// TIA Portal V15.1 export
// export: Created 2024-06-21T08:40:57.1284392Z, ExportSetting WithDefaults, DisplayName Totally Integrated Automation Portal, DisplayVersion V15.1 Update 5, DisplayName TIA Portal Openness, DisplayVersion V15.1 Update 5, DisplayName SINAMICS Startdrive Advanced, DisplayVersion V15.1, DisplayName G130, G150, S120, S150, SINAMICS MV, S210, DisplayVersion V15.1, DisplayName G110M, G120, G120C, G120D, G120P, DisplayVersion V15.1, DisplayName STEP 7 Professional, DisplayVersion V15.1 Update 5, DisplayName STEP 7 Safety, DisplayVersion V15.1, DisplayName WinCC Professional, DisplayVersion V15.1 Update 5, DisplayName SIMATIC Visualization Architect, DisplayVersion V15.1
FUNCTION_BLOCK "L1SafetyFbkAlarm"   // FB1422, FBD
TITLE = L1SafetyFbkAlarm
{ S7_Optimized_Access := 'FALSE' }
AUTHOR : VCC
FAMILY : AlarmHnd
NAME : 1SafeAlm
VERSION : 0.3
// ================================================================================
// TThis module evalute the diagnostic byte from the Siemens safety Functionblock 
// FB 216 "F_FDBACK" and generates a feedback alarm in the standard program.
// A boolean output is available to inform the upper level that the alarm can be 
// reset.
// This module generates also a word containing all necessary information for HMI 
// Icon animation, and a word with all information for HMI safety module 
// diagnostic screen. 
// ================================================================================
// stored: AutoNumber false, IsIECCheckEnabled false, SetENOAutomatically False, UDAEnableTagReadback false
   VAR_INPUT
      I_Feedback { ExternalAccessible := 'False'; ExternalVisible := 'False'; ExternalWritable := 'False'} : Bool;   // Input feedback
      I_AlarmClass { ExternalAccessible := 'False'; ExternalVisible := 'False'; ExternalWritable := 'False'} : Char;   // Alarm class -> A - B - C - D or E
      I_EnableAlarm { ExternalAccessible := 'False'; ExternalVisible := 'False'; ExternalWritable := 'False'} : Bool := TRUE;   // Enable alarm from upper level (0=disable/1=enable)
      I_AlarmResetPB { ExternalAccessible := 'False'; ExternalVisible := 'False'; ExternalWritable := 'False'} : Bool;   // Alarm reset pushbutton is activated
      I_SafetyCard_DIAG { ExternalAccessible := 'False'; ExternalVisible := 'False'; ExternalWritable := 'False'} : Byte;   // Automatically generated DB from F-Modul (F-Peripherie DB)
   END_VAR
   VAR_OUTPUT
      O_Alarm { ExternalAccessible := 'False'; ExternalVisible := 'False'; ExternalWritable := 'False'} : Bool;   // Alarm
      O_AlarmABCondiion { ExternalAccessible := 'False'; ExternalVisible := 'False'; ExternalWritable := 'False'} : Bool;   // Alarm AB condition
      H_IAnim { ExternalAccessible := 'False'; ExternalVisible := 'False'; ExternalWritable := 'False'} : Word;   // Icon Animation
   END_VAR
   VAR DB_SPECIFIC
      H_Out : Struct   // HMI
         Anim : Word;   // HMI Animation of the object
         DBnr : Int;   // HMI Animation DB number
      END_STRUCT;
      FeedbackError { ExternalAccessible := 'False'; ExternalVisible := 'False'; ExternalWritable := 'False'} : Bool;   // Feedback error or incorrect feedback time setting (= state of ERROR)
      Passivation { ExternalAccessible := 'False'; ExternalVisible := 'False'; ExternalWritable := 'False'} : Bool;   // Passivation of F-I/O/channel controlled by output Q
      ErrorSignal0 { ExternalAccessible := 'False'; ExternalVisible := 'False'; ExternalWritable := 'False'} : Bool;   // After feedback error: feedback input has permanent signal state of 0
      ErrorSignal1 { ExternalAccessible := 'False'; ExternalVisible := 'False'; ExternalWritable := 'False'} : Bool;   // For feedback error: input ACK has a permanent signal state of 1
      AckReq { ExternalAccessible := 'False'; ExternalVisible := 'False'; ExternalWritable := 'False'} : Bool;   // Acknowledgement required (= state of ACK_REQ)
      Q { ExternalAccessible := 'False'; ExternalVisible := 'False'; ExternalWritable := 'False'} : Bool;   // State of output Q
      Alarm { ExternalAccessible := 'False'; ExternalVisible := 'False'; ExternalWritable := 'False'} : Bool;   // Alarm
      AlarmClass_A { ExternalAccessible := 'False'; ExternalVisible := 'False'; ExternalWritable := 'False'} : Bool;   // The alarm is from alarm class A
      AlarmClass_B { ExternalAccessible := 'False'; ExternalVisible := 'False'; ExternalWritable := 'False'} : Bool;   // The alarm is from alarm class B
      AlarmClass_C { ExternalAccessible := 'False'; ExternalVisible := 'False'; ExternalWritable := 'False'} : Bool;   // The alarm is from alarm class C
      AlarmClass_D { ExternalAccessible := 'False'; ExternalVisible := 'False'; ExternalWritable := 'False'} : Bool;   // The alarm is from alarm class D
      AlarmCond { ExternalAccessible := 'False'; ExternalVisible := 'False'; ExternalWritable := 'False'} : Bool;   // Alarm condition
      DBnr { ExternalAccessible := 'False'; ExternalVisible := 'False'; ExternalWritable := 'False'} : Int;   // HMI DB number
   END_VAR
BEGIN

NETWORK
TITLE = **** 1 - Inputs **** DB number
// DB number
      L     DINO;
      T     #DBnr;

NETWORK
TITLE = **** 1 - Inputs **** Alarm class
// Alarm class
// Alarm class = D
      L     #I_AlarmClass;
      L     'D';
      ==I;
      =     #AlarmClass_D;

// Alarm class = C
      L     #I_AlarmClass;
      L     'C';
      ==I;
      =     #AlarmClass_C;

// Alarm class = B
      L     #I_AlarmClass;
      L     'B';
      ==I;
      =     #AlarmClass_B;

// Alarm class = A
      AN    #AlarmClass_B;
      AN    #AlarmClass_C;
      AN    #AlarmClass_D;
      =     #AlarmClass_A;


REGION Network 3: **** 1 - Inputs **** Feedback error or incorrect feedback time setting (= state of ERROR)
   // Feedback error or incorrect feedback time setting (= state of ERROR)
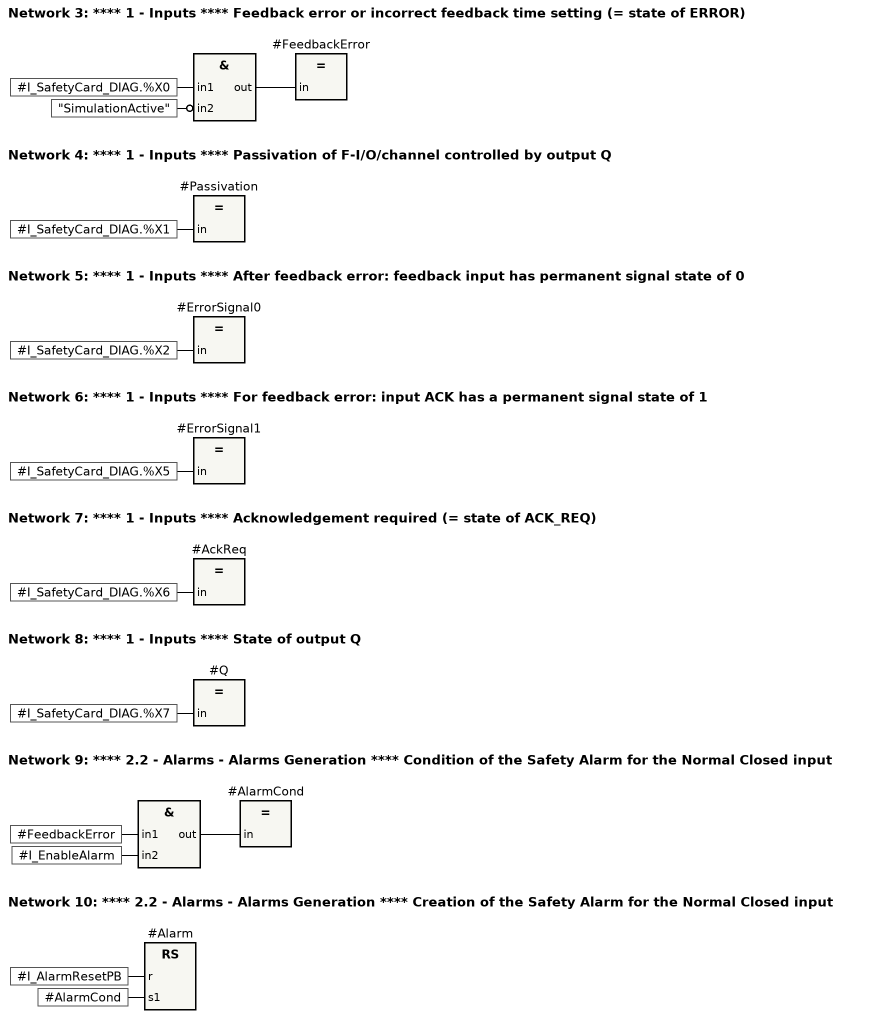
   #FeedbackError := #I_SafetyCard_DIAG.%X0 AND NOT "SimulationActive";
END_REGION

REGION Network 4: **** 1 - Inputs **** Passivation of F-I/O/channel controlled by output Q
   // Passivation of F-I/O/channel controlled by output Q
   #Passivation := #I_SafetyCard_DIAG.%X1;
END_REGION

REGION Network 5: **** 1 - Inputs **** After feedback error: feedback input has permanent signal state of 0
   // After feedback error: feedback input has permanent signal state of 0
   #ErrorSignal0 := #I_SafetyCard_DIAG.%X2;
END_REGION

REGION Network 6: **** 1 - Inputs **** For feedback error: input ACK has a permanent signal state of 1
   // For feedback error: input ACK has a permanent signal state of 1
   #ErrorSignal1 := #I_SafetyCard_DIAG.%X5;
END_REGION

REGION Network 7: **** 1 - Inputs **** Acknowledgement required (= state of ACK_REQ)
   // Acknowledgement required (= state of ACK_REQ)
   #AckReq := #I_SafetyCard_DIAG.%X6;
END_REGION

REGION Network 8: **** 1 - Inputs **** State of output Q
   // State of output Q
   #Q := #I_SafetyCard_DIAG.%X7;
END_REGION

REGION Network 9: **** 2.2 - Alarms - Alarms Generation **** Condition of the Safety Alarm for the Normal Closed input
   // Condition of the Safety Alarm for the Normal Closed input
   #AlarmCond := #FeedbackError AND #I_EnableAlarm;
END_REGION

REGION Network 10: **** 2.2 - Alarms - Alarms Generation **** Creation of the Safety Alarm for the Normal Closed input
   // Creation of the Safety Alarm for the Normal Closed input
   IF #I_AlarmResetPB THEN
       #Alarm := FALSE;   // RS flip-flop
   END_IF;
   IF #AlarmCond THEN #Alarm := TRUE; END_IF;
END_REGION

REGION Network 11: **** 4.6 - Mashine Status - Indications **** Icon Animation
   // Icon Animation
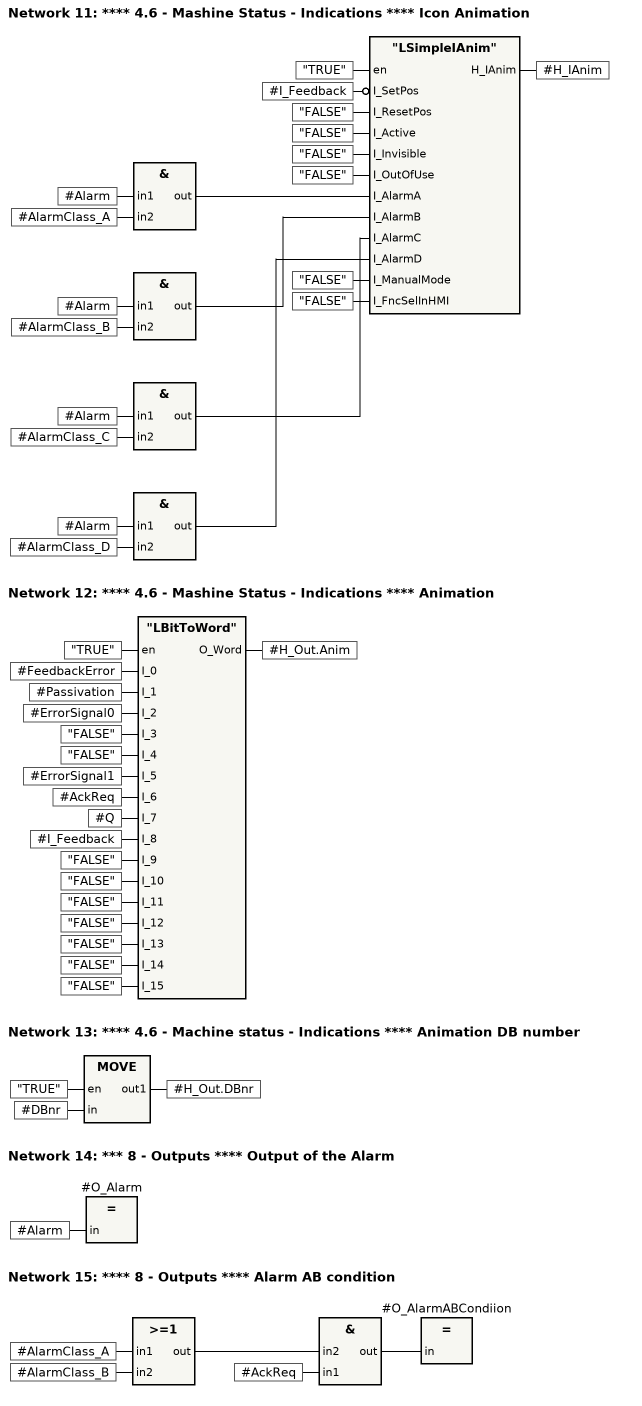
   IF "TRUE" THEN
       "LSimpleIAnim"(I_SetPos := NOT #I_Feedback,
                      I_ResetPos := "FALSE",
                      I_Active := "FALSE",
                      I_Invisible := "FALSE",
                      I_OutOfUse := "FALSE",
                      I_AlarmA := #Alarm AND #AlarmClass_A,
                      I_AlarmB := #Alarm AND #AlarmClass_B,
                      I_AlarmC := #Alarm AND #AlarmClass_C,
                      I_AlarmD := #Alarm AND #AlarmClass_D,
                      I_ManualMode := "FALSE",
                      I_FncSelInHMI := "FALSE",
                      H_IAnim => #H_IAnim);
   END_IF;
END_REGION

REGION Network 12: **** 4.6 - Mashine Status - Indications **** Animation
   // Animation
   IF "TRUE" THEN
       "LBitToWord"(I_0 := #FeedbackError,
                    I_1 := #Passivation,
                    I_2 := #ErrorSignal0,
                    I_3 := "FALSE",
                    I_4 := "FALSE",
                    I_5 := #ErrorSignal1,
                    I_6 := #AckReq,
                    I_7 := #Q,
                    I_8 := #I_Feedback,
                    I_9 := "FALSE",
                    I_10 := "FALSE",
                    I_11 := "FALSE",
                    I_12 := "FALSE",
                    I_13 := "FALSE",
                    I_14 := "FALSE",
                    I_15 := "FALSE",
                    O_Word => #H_Out.Anim);
   END_IF;
END_REGION

REGION Network 13: **** 4.6 - Machine status - Indications **** Animation DB number
   // Animation DB number
   IF "TRUE" THEN #H_Out.DBnr := #DBnr; END_IF;
END_REGION

REGION Network 14: *** 8 - Outputs **** Output of the Alarm
   // Output of the Alarm
   #O_Alarm := #Alarm;
END_REGION

REGION Network 15: **** 8 - Outputs **** Alarm AB condition
   // Alarm AB condition
   #O_AlarmABCondiion := (#AlarmClass_A OR #AlarmClass_B) AND #AckReq;
END_REGION
END_FUNCTION_BLOCK
